// TwinCAT 3 PLC project CX7080
// ProgramVersion: 3.1.4024.0
// libraries:
//   Tc2_Standard, * (Beckhoff Automation GmbH)
//   Tc2_System, * (Beckhoff Automation GmbH)
//   Tc3_Module, * (Beckhoff Automation GmbH)
// project tree:
//   DUTs/ state_enum.TcDUT
//   / GlobalTextList.TcGTLO, PlcTask.TcTTO, Visualization Manager.TcVMO (not stored)
//   GVLs/ GVL.TcGVL
//   POUs/ FB_Auto.TcPOU, FB_Comm_Fault.TcPOU, FB_Emg_Stop.TcPOU, FB_Jog_Cartesian.TcPOU, FB_Jog_Joint.TcPOU, FB_Manual.TcPOU, FB_ModbusComm.TcPOU, FB_Startup.TcPOU, main_prg.TcPOU
// real-time tasks:
//   TASK PlcTask: cycle T#10ms, priority 20, ADS port 350

CONFIGURATION CX7080
    RESOURCE PLC ON TwinCAT3
        TASK PlcTask(INTERVAL := T#10ms, PRIORITY := 21);
        PROGRAM main_prg WITH PlcTask : main_prg;
    END_RESOURCE
END_CONFIGURATION

// ---- DUTs/state_enum.TcDUT
{attribute 'qualified_only'}
{attribute 'strict'}
TYPE state_enum :
(
	startup_mode,
	jog_joint_mode,
	jog_cartesian_mode,
	auto_mode,
	emg_stop_mode,
	comm_fault_mode,
	manual_mode
);
END_TYPE

// ---- GVLs/GVL.TcGVL
{attribute 'qualified_only'}
VAR_GLOBAL
	// Internal system parameters
	system_state : state_enum := state_enum.startup_mode; // Used to keep track of system state machine. Initialized in startup_mode.
	modbus_comm_fault : BOOL := FALSE;
	J1_Home_Pos : INT := 135; // Degrees
	J2_Home_Pos : INT := 135; // Degrees
	J3_Home_Pos : INT := 135; // Degrees
	J1_Value : INT := 135;
	J2_Value : INT := 135;
	J3_Value : INT := 135;
	
	// Inputs
	input1 AT %I* : BOOL;
	output1 AT %Q* : BOOL;
	PB_J1_CW AT %I* : BOOL;
	PB_J1_CCW AT %I*: BOOL;
	PB_J2_CW AT %I* : BOOL;
	PB_J2_CCW AT %I* : BOOL;
	PB_J3_CW AT %I* : BOOL;
	PB_J3_CCW AT %I* : BOOL;
	PB_EE_Grip AT %I* : BOOL;
	PB_EE_Ungrip AT %I* : BOOL;
	PB_EMG_STOP AT %I* : BOOL;
	PB_Reset AT %I* : BOOL;
	PB_Record_Pos AT %I* : BOOL;
	PB_Record_Delay AT %I* : BOOL;
	PB_Start_Pause AT %I* : BOOL;
	SW_Slow_Fast AT %I* : BOOL;
	SW_Join_Cart AT %I* : BOOL;
	
	// Outputs
	LED_J1_CW AT %Q* : BOOL;
	LED_J1_CCW AT %Q*: BOOL;
	LED_J2_CW AT %Q* : BOOL;
	LED_J2_CCW AT %Q* : BOOL;
	LED_J3_CW AT %Q* : BOOL;
	LED_J3_CCW AT %Q* : BOOL;
	LED_EE_Grip AT %Q* : BOOL;
	LED_EE_Ungrip AT %Q* : BOOL;
	LED_EMG_STOP AT %Q* : BOOL;
	LED_Reset AT %Q* : BOOL;
	LED_Record_Pos AT %Q* : BOOL;
	LED_Record_Delay AT %Q* : BOOL;
	LED_Start_Pause AT %Q* : BOOL;
	LED_Comm_Fault AT %Q* : BOOL;
	LED_Warning AT %Q* : BOOL;
	
	// Modbus registers
	MB_Write_J1 : INT;
	MB_Write_J2 : INT;
	MB_Write_J3 : INT;
	MB_Write_Gripper : INT;
	MB_Write_Watchdog : INT;
	MB_Write_Blank1 : INT;
	MB_Write_Blank2 : INT;
	MB_Write_Blank3 : INT;
	MB_Write_Blank4 : INT;
	MB_Write_Blank5 : INT;
	MB_Read_Watchdog : INT;
	MB_Read_Blank2 : INT;
	MB_Read_Blank3 : INT;
	MB_Read_Blank4 : INT;
	MB_Read_Blank5 : INT;
	MB_Read_Blank6 : INT;
	MB_Read_Blank7 : INT;
	MB_Read_Blank8 : INT;
	MB_Read_Blank9 : INT;
	MB_Read_Blank10 : INT;
END_VAR

// ---- POUs/main_prg.TcPOU
PROGRAM main_prg
VAR
	last_state : state_enum;
	fb_Startup : FB_Startup;
	fb_Auto : FB_Auto;
	fb_Comm_Fault : FB_Comm_Fault;
	fb_Emg_Stop : FB_Emg_Stop;
	fb_Jog_Cartesian : FB_Jog_Cartesian;
	fb_Jog_Joint : FB_Jog_Joint;
	fb_Manual : FB_Manual;
	fb_ModbusComm : FB_ModbusComm;
END_VAR

IF NOT GVL.PB_EMG_STOP AND NOT (gvl.system_state = state_enum.startup_mode) THEN
	GVL.system_state := state_enum.emg_stop_mode;
ELSIF GVL.modbus_comm_fault AND NOT (gvl.system_state = state_enum.startup_mode)  THEN
	GVL.system_state := state_enum.comm_fault_mode;
END_IF


CASE gvl.system_state OF
state_enum.startup_mode:
	fb_Startup();
state_enum.jog_joint_mode:
	fb_Jog_Joint();
state_enum.jog_cartesian_mode:
	fb_Jog_Cartesian();
state_enum.manual_mode:
	fb_Manual();
state_enum.emg_stop_mode:
	fb_Emg_Stop();
state_enum.comm_fault_mode:
	fb_Comm_Fault();
state_enum.auto_mode:
	fb_Auto();
END_CASE

fb_ModbusComm();

END_PROGRAM

// ---- POUs/FB_Startup.TcPOU
FUNCTION_BLOCK FB_Startup
VAR_INPUT
END_VAR
VAR_OUTPUT
END_VAR
VAR
	timer1 : TON;
	timer2 : TON;
	timer3 : TON;
	timer4 : TON;
	timer5 : TON;
	timer6 : TON;
	timer7 : TON;
	EMG_STOP_RELEASED : BOOL;
END_VAR

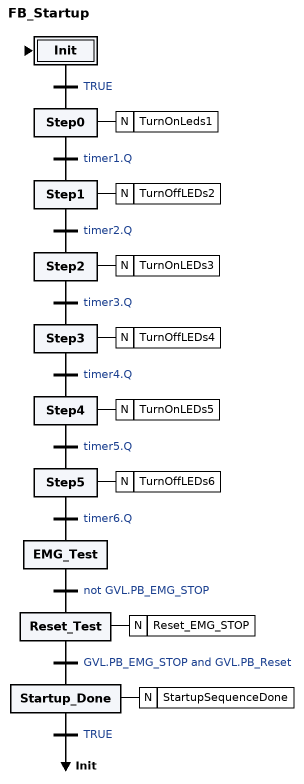
INITIAL_STEP Init:
END_STEP
TRANSITION FROM Init TO Step0
    := TRUE;
END_TRANSITION
STEP Step0:
    TurnOnLeds1(N);
END_STEP
TRANSITION FROM Step0 TO Step1
    := timer1.Q;
END_TRANSITION
STEP Step1:
    TurnOffLEDs2(N);
END_STEP
TRANSITION FROM Step1 TO Step2
    := timer2.Q;
END_TRANSITION
STEP Step2:
    TurnOnLEDs3(N);
END_STEP
TRANSITION FROM Step2 TO Step3
    := timer3.Q;
END_TRANSITION
STEP Step3:
    TurnOffLEDs4(N);
END_STEP
TRANSITION FROM Step3 TO Step4
    := timer4.Q;
END_TRANSITION
STEP Step4:
    TurnOnLEDs5(N);
END_STEP
TRANSITION FROM Step4 TO Step5
    := timer5.Q;
END_TRANSITION
STEP Step5:
    TurnOffLEDs6(N);
END_STEP
TRANSITION FROM Step5 TO EMG_Test
    := timer6.Q;
END_TRANSITION
STEP EMG_Test:
END_STEP
TRANSITION FROM EMG_Test TO Reset_Test
    := not GVL.PB_EMG_STOP;
END_TRANSITION
STEP Reset_Test:
    Reset_EMG_STOP(N);
END_STEP
TRANSITION FROM Reset_Test TO Startup_Done
    := GVL.PB_EMG_STOP and GVL.PB_Reset;
END_TRANSITION
STEP Startup_Done:
    StartupSequenceDone(N);
END_STEP
TRANSITION FROM Startup_Done TO Init
    := TRUE;
END_TRANSITION

METHOD AllLEDsTrigger : BOOL
VAR_INPUT
	OnOff : BOOL; // OnOff - Turn off, True - Turn On
END_VAR
GVL.LED_Comm_Fault := OnOff;
GVL.LED_EE_Grip := OnOff;
GVL.LED_EE_Ungrip := OnOff;
GVL.LED_EMG_STOP := OnOff;
GVL.LED_J1_CCW := OnOff;
GVL.LED_J1_CW := OnOff;
GVL.LED_J2_CCW := OnOff;
GVL.LED_J2_CW := OnOff;
GVL.LED_J3_CCW := OnOff;
GVL.LED_J3_CW := OnOff;
GVL.LED_Record_Delay := OnOff;
GVL.LED_Record_Pos := OnOff;
GVL.LED_Reset := OnOff;
GVL.LED_Start_Pause := OnOff;
GVL.LED_Warning := OnOff;
END_METHOD

ACTION Reset_EMG_STOP:
IF NOT GVL.PB_EMG_STOP THEN
	GVL.LED_EMG_STOP := TRUE;
END_IF

IF GVL.PB_EMG_STOP THEN
	GVL.LED_EMG_STOP := FALSE;
	GVL.LED_Reset := TRUE;
END_IF
END_ACTION

ACTION StartupSequenceDone:
GVL.LED_EMG_STOP := FALSE;
GVL.LED_Reset := FALSE;
GVL.system_state := state_enum.jog_joint_mode;
END_ACTION

ACTION TurnOffLEDs2:
timer1(IN := FALSE, PT := T#1S);
timer2(IN := TRUE, PT := T#1S);
timer3(IN := FALSE, PT := T#1S);
timer4(IN := FALSE, PT := T#1S);
timer5(IN := FALSE, PT := T#1S);
timer6(IN := FALSE, PT := T#1S);
timer7(IN := FALSE, PT := T#1S);
AllLEDsTrigger(FALSE);
END_ACTION

ACTION TurnOffLEDs4:
timer1(IN := FALSE, PT := T#1S);
timer2(IN := FALSE, PT := T#1S);
timer3(IN := FALSE, PT := T#1S);
timer4(IN := TRUE, PT := T#1S);
timer5(IN := FALSE, PT := T#1S);
timer6(IN := FALSE, PT := T#1S);
timer7(IN := FALSE, PT := T#1S);
AllLEDsTrigger(FALSE);
END_ACTION

ACTION TurnOffLEDs6:
timer1(IN := FALSE, PT := T#1S);
timer2(IN := FALSE, PT := T#1S);
timer3(IN := FALSE, PT := T#1S);
timer4(IN := FALSE, PT := T#1S);
timer5(IN := FALSE, PT := T#1S);
timer6(IN := TRUE, PT := T#1S);
timer7(IN := FALSE, PT := T#1S);
AllLEDsTrigger(FALSE);
END_ACTION

ACTION TurnOnLeds1:
timer1(IN := TRUE, PT := T#1S);
timer2(IN := FALSE, PT := T#1S);
timer3(IN := FALSE, PT := T#1S);
timer4(IN := FALSE, PT := T#1S);
timer5(IN := FALSE, PT := T#1S);
timer6(IN := FALSE, PT := T#1S);
timer7(IN := FALSE, PT := T#1S);
AllLEDsTrigger(TRUE);
END_ACTION

ACTION TurnOnLEDs3:
timer1(IN := FALSE, PT := T#1S);
timer2(IN := FALSE, PT := T#1S);
timer3(IN := TRUE, PT := T#1S);
timer4(IN := FALSE, PT := T#1S);
timer5(IN := FALSE, PT := T#1S);
timer6(IN := FALSE, PT := T#1S);
timer7(IN := FALSE, PT := T#1S);
AllLEDsTrigger(TRUE);
END_ACTION

ACTION TurnOnLEDs5:
timer1(IN := TRUE, PT := T#1S);
timer2(IN := FALSE, PT := T#1S);
timer3(IN := FALSE, PT := T#1S);
timer4(IN := FALSE, PT := T#1S);
timer5(IN := TRUE, PT := T#1S);
timer6(IN := FALSE, PT := T#1S);
timer7(IN := FALSE, PT := T#1S);
AllLEDsTrigger(TRUE);
END_ACTION

END_FUNCTION_BLOCK

// ---- POUs/FB_Auto.TcPOU
FUNCTION_BLOCK FB_Auto
VAR_INPUT
END_VAR
VAR_OUTPUT
END_VAR
VAR
END_VAR

END_FUNCTION_BLOCK

// ---- POUs/FB_Comm_Fault.TcPOU
FUNCTION_BLOCK FB_Comm_Fault
VAR_INPUT
END_VAR
VAR_OUTPUT
END_VAR
VAR
END_VAR

END_FUNCTION_BLOCK

// ---- POUs/FB_Emg_Stop.TcPOU
FUNCTION_BLOCK FB_Emg_Stop
VAR_INPUT
END_VAR
VAR_OUTPUT
END_VAR
VAR
	fb_Blink_Reset: FB_Blink;
	resetPushTime : TIME := T#3S;
	resetBlinkOnTime : TIME := T#500ms;
	resetTimer: TON;
END_VAR

IF NOT GVL.PB_EMG_STOP THEN
	GVL.LED_EMG_STOP := TRUE;
	GVL.LED_Reset := FALSE;
ELSE
	GVL.LED_EMG_STOP := FALSE;
END_IF

IF GVL.PB_EMG_STOP AND NOT GVL.PB_Reset THEN
	GVL.LED_EMG_STOP := TRUE;
ELSE
	GVL.LED_EMG_STOP := FALSE;
END_IF

IF GVL.PB_EMG_STOP AND GVL.PB_Reset THEN
	resetTimer(IN:= GVL.PB_Reset, PT:= resetPushTime, Q=> , ET=> );
END_IF;

IF GVL.PB_Reset AND NOT resetTimer.Q THEN
	fb_Blink_Reset(OnOffTime:= resetBlinkOnTime, TriggerBlink:= TRUE, BlinkSignal=> GVL.LED_Reset);
ELSIF GVL.PB_Reset AND resetTimer.Q THEN
	fb_Blink_Reset(OnOffTime:= resetBlinkOnTime, TriggerBlink:= FALSE, BlinkSignal=> GVL.LED_Reset);
	GVL.LED_Reset := FALSE;
	GVL.system_state := state_enum.auto_mode; // TODO: Should change back to last state, not auto_mode
END_IF;

END_FUNCTION_BLOCK

// ---- POUs/FB_Jog_Cartesian.TcPOU
FUNCTION_BLOCK FB_Jog_Cartesian
VAR_INPUT
	X : REAL;
	Y : REAL;
	Z : REAL;
	L1 : REAL;
	L2 : REAL;
	L3 : REAL;
	
END_VAR
VAR_OUTPUT
	OutputBaseAngle : INT;
	OutputShoulderAngle : INT;
	OutputElbowAngle : INT;
END_VAR

VAR
END_VAR

//		     GOTTA GO CARTESIAN
//              ___------__
//        |\__-- /\       _-
//        |/    __      -
//        //\  /  \    /__
//        |  o|  0|__     --_
//        \\____-- __ \   ___-
//        (@@    __/  / /_
//           -_____---   --_
//            //  \ \\   ___-
//          //|\__/  \\  \
//          \_-\_____/  \-\
//               // \\--\|   
//          ____//  ||_
//         /_____\ /___\
//       ______________________⠀⠀

OutputBaseAngle := REAL_TO_INT(L1 * TAN(X));
OutputShoulderAngle := REAL_TO_INT(L2 * SIN(Y));
OutputElbowAngle := REAL_TO_INT(L3 * COS(Z));

END_FUNCTION_BLOCK

// ---- POUs/FB_Jog_Joint.TcPOU
FUNCTION_BLOCK FB_Jog_Joint
VAR_INPUT
	StopServos : BOOL;
	RampSpeedSetting : BOOL; // False : Low speed, True: High speed
	BaseIncreaseCW : BOOL;
	BaseIncreaseCCW : BOOL;
	ShoulderIncreaseCW : BOOL;
	ShoulderIncreaseCCW : BOOL;
	ElbowIncreaseCW : BOOL;
	ElbowIncreaseCCW : BOOL;
	RampSpeedLow : REAL;
	RampSpeedHigh : REAL;
	BaseAngleMin : INT;
	BaseAngleMax : INT;
	ShoulderAngleMin : INT;
	ShoulderAngleMax : INT;
	ElbowAngleMin : INT;
	ElbowAngleMax : INT;
	RampCycleTime : TIME; // Must be the same as task cycle time
	BaseStartPos : INT;
	ShoulderStartPos : INT;
	ElbowStartPos : INT;
END_VAR
VAR_OUTPUT
	BaseServoOutput : INT;
	ShoulderServoOutput : INT;
	ElbowServoOutput : INT;
END_VAR
VAR
	fb_Base_Servo: FB_RC_Servo;
	fb_ElbowServo: FB_RC_Servo;
	fb_ShoulderServo: FB_RC_Servo;
	CurrentSpeedSetting : REAL;
	BaseSetpoint : INT;
	ShoulderSetpoint : INT;
	ElbowSetpoint : INT;
END_VAR

IF RampSpeedSetting THEN
	CurrentSpeedSetting := RampSpeedHigh;
ELSE
	CurrentSpeedSetting := RampSpeedLow;
END_IF

IF BaseIncreaseCW AND NOT BaseIncreaseCCW THEN
	BaseSetpoint := BaseAngleMin;
ELSIF NOT BaseIncreaseCW AND BaseIncreaseCCW THEN
	BaseSetpoint := BaseAngleMax;
ELSIF NOT BaseIncreaseCW AND NOT BaseIncreaseCCW THEN
	BaseSetpoint := BaseServoOutput;
END_IF

IF ShoulderIncreaseCW AND NOT ShoulderIncreaseCCW THEN
	ShoulderSetpoint := ShoulderAngleMin;
ELSIF NOT ShoulderIncreaseCW AND ShoulderIncreaseCCW THEN
	ShoulderSetpoint := ShoulderAngleMax;
ELSIF NOT ShoulderIncreaseCW AND NOT ShoulderIncreaseCCW THEN
	ShoulderSetpoint := ShoulderServoOutput;
END_IF

IF ElbowIncreaseCW AND NOT ElbowIncreaseCCW THEN
	ElbowSetpoint := ElbowAngleMin;
ELSIF NOT ElbowIncreaseCW AND ElbowIncreaseCCW THEN
	ElbowSetpoint := ElbowAngleMax;
ELSIF NOT ElbowIncreaseCW AND NOT ElbowIncreaseCCW THEN
	ElbowSetpoint := ElbowServoOutput;
END_IF


fb_Base_Servo(
	stop:= StopServos, 
	setpoint:= BaseSetpoint, 
	rampSpeed:= CurrentSpeedSetting, 
	trapezoidalProfileActive:= , 
	servoAngleMin:= BaseAngleMin, 
	servoAngleMax:= BaseAngleMax, 
	rampCycleTime:= RampCycleTime, 
	rampStartPos:= BaseStartPos, 
	currentPositionSetpoint=> BaseServoOutput, 
	error=> );

	
fb_ShoulderServo(
	stop:= StopServos, 
	setpoint:= ShoulderSetpoint, 
	rampSpeed:= CurrentSpeedSetting, 
	trapezoidalProfileActive:= , 
	servoAngleMin:= ShoulderAngleMin, 
	servoAngleMax:= ShoulderAngleMax, 
	rampCycleTime:= RampCycleTime, 
	rampStartPos:= ShoulderStartPos, 
	currentPositionSetpoint=> ShoulderServoOutput, 
	error=> );
	
	
fb_ElbowServo(
	stop:= StopServos, 
	setpoint:= ElbowSetpoint, 
	rampSpeed:= CurrentSpeedSetting, 
	trapezoidalProfileActive:= , 
	servoAngleMin:= ElbowAngleMin, 
	servoAngleMax:= ElbowAngleMax, 
	rampCycleTime:= RampCycleTime, 
	rampStartPos:= ElbowStartPos, 
	currentPositionSetpoint=> ElbowServoOutput, 
	error=> );

END_FUNCTION_BLOCK

// ---- POUs/FB_Manual.TcPOU
FUNCTION_BLOCK FB_Manual
VAR_INPUT
END_VAR
VAR_OUTPUT
END_VAR
VAR
END_VAR

END_FUNCTION_BLOCK

// ---- POUs/FB_ModbusComm.TcPOU
FUNCTION_BLOCK FB_ModbusComm
VAR_INPUT
END_VAR
VAR_OUTPUT
END_VAR
VAR
END_VAR

END_FUNCTION_BLOCK
